# EPICS autosave request: src/NDPluginGeometricTransform/NDGeometricTransform_settings.req
$(P)$(R)EnableScaling
